(* CoDeSys 2.3 library: Visu_Scheduler_02_F.lib *)
(* Libraries: Standard.lib 4.10.05 11:14:46, SYSLIBCALLBACK.LIB 20.4.05 10:04:48 *)

(* POU French_PublicHoliday, ST *)
FUNCTION_BLOCK French_PublicHoliday
VAR
	Init:BOOL:=TRUE;
END_VAR

VAR_IN_OUT
	typPublicHoliday:typPublicHoliday;
END_VAR
VAR_INPUT
	EN:BOOL;
END_VAR
IF EN AND INIT THEN

(*8 mai*)
typPublicHoliday.SpecialPublicHoliday1_day:=8;
typPublicHoliday.SpecialPublicHoliday1_month:=5;

(*14 juillet*)
typPublicHoliday.SpecialPublicHoliday2_day:=14;
typPublicHoliday.SpecialPublicHoliday2_month:=7;

(*11 novembre*)
typPublicHoliday.SpecialPublicHoliday1_day:=11;
typPublicHoliday.SpecialPublicHoliday1_month:=11;

Init:=FALSE;

END_IF
END_FUNCTION_BLOCK
